(* CODESYS project myRepo003

Project tree, tasks and I/O mapping:
  Device : 750-8212 PFC200, WAGO, order no. 750-8212, version 6.0.0.15
    application Application
      libraries: Standard, * (System)
      task MainTask (cyclic, interval t#50ms, priority 15) calls PLC_PRG
      program PLC_PRG [ST]
    Kbus : Kbus, WAGO, version 2.1.0.1
        unmapped channels: K-BUS diagnostics
      _750_469_003_000_04 : 750-469/003-000#04, WAGO, order no. 750-469/003-000, version 2.0.0.9
          unmapped channels: _IINT 1, _IINT 2
      _750_494_24 : 750-494#24, WAGO, order no. 750-494, version 2.0.0.24
          unmapped channels: _ST, _IN, _CTL, _NOT_USED
      _75x_2DI : 75x-2DI, WAGO, version 2.0.0.13
          unmapped channels: _IN
      _75x_2DO : 75x-2DO, WAGO, version 2.0.0.13
          output dq : BYTE  // _OUT
    Serial
      COM1 : COM1, WAGO, version 0.0.0.19
*)

// Device/Application/PLC_PRG
PROGRAM PLC_PRG
VAR
END_VAR

dq:=dq+1;

END_PROGRAM
